ABB RobotStudio station: p3_robotstudio_2parte_ampliacion.rspag

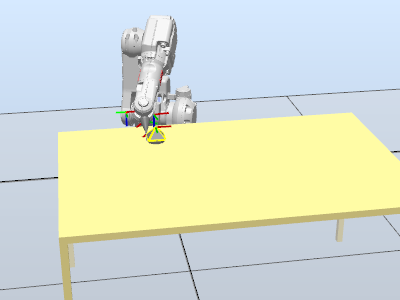
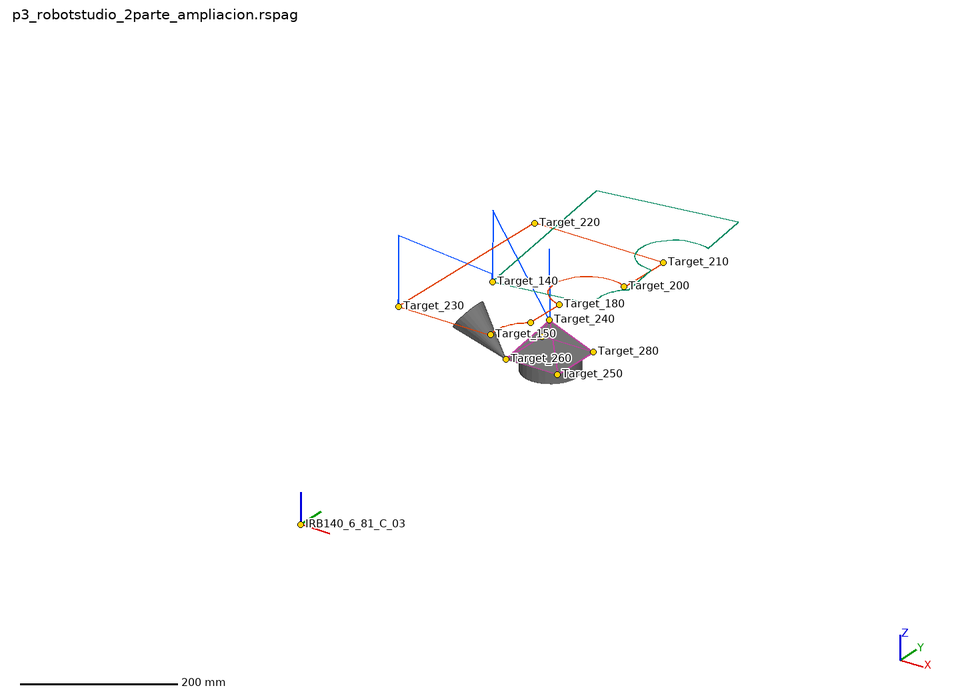
[picture v1: parts stored in the station drawn from their meshes, with robot base, taught points and paths (robot models come from the ABB library and are not in the file)]
--- station ---
Station p3_robotstudio_2parte (saved by RobotStudio 22.2.10013.1)
Controller Controlador1
  mechanical unit ROB_1: IRB140_6_81_C_03, 6 joints, base frame (0, 0, 0) mm
Layout (positions relative to the parent item):
  - printbed_hemisphere_hexagono [part, from Libraries\hemisphere.rslib] at (471.3, 85, 364.75) mm, rotated rx 90 ry 0 rz 0 deg
  - Mesa de trabajo [part, from Libraries\Mesa de trabajoDISA.rslib] at (1242.15, -525.68, -395) mm, rotated rx 0 ry 0 rz 90 deg
  - Pieza1 [part, from Libraries\Pieza_ampliacion.rslib] at (500, 0, 200) mm, rotated rx 0 ry 0 rz 90 deg
  - trazador [smart component, from Libraries\trazador.rslib] at (335.01, -108.97, 433.65) mm, rotated rx -146.48 ry 41.47 rz -135 deg
      connections:
        trazador.entrada_inyector -> TraceTCP.Enabled
        trazador.entrada_inyector -> ?.InputA
        ?.Output -> TraceTCP.Clear
    - TraceTCP [smart component, from Components\TraceTCP.rslib]
        properties: Robot=IRB140_6_81_C_03
  - IRB140_6_81_C_03 [mechanism, from Robots\IRB140_6_81_C_G_03.rslib] at (0, 0, 0) mm; joint values [-0.3661, -0.187, 0.842, 1.3893, 0.2881, -2.1751] (rad or m)
  - tool_laser [part] at (335.01, -108.97, 433.65) mm, rotated rx -146.48 ry 41.47 rz -135 deg, size 50 x 49.9 x 75 mm
  - tool_laser [mechanism] at (335.01, -108.97, 433.65) mm, rotated rx -146.48 ry 41.47 rz -135 deg
      TCP tool_laser at (0, 0, 75) mm
      links: Pieza_1
  - Curve_thing [part, from Training Objects\Curve_Thing.rslib] at (542.09, -125.55, 364.72) mm, rotated rx 0 ry 0.37 rz 89.92 deg
  - Pieza_4 [part] at (610.67, 44.58, 426.77) mm
  - Pieza_8 [part] at (-348.26, -126.32, -48.58) mm, size 80.8 x 80.4 x 70 mm
Attachment: trazador is attached to IRB140_6_81_C_03 / Link6
Attachment: tool_laser is attached to IRB140_6_81_C_03 / Link6
Attachment: tool_laser is attached to IRB140_6_81_C_03 / Link6
Attachment: Curve_thing is attached to Mesa de trabajo
Station logic (signal -> signal, property => property):
  Controlador1.activar_mecanizado -> trazador.entrada_inyector
Targets, tools, work objects and paths stored in the station and not in the controller backup, written as RAPID:
! task T_ROB1
MODULE Module1
  CONST robtarget Target_300:=[[-0.030300341,0.033376716,-0.180784391],[0.786632811,0.381173416,0.211660446,-0.437167591],[0,0,0,0],[9E+09,9E+09,9E+09,9E+09,9E+09,9E+09]];
ENDMODULE


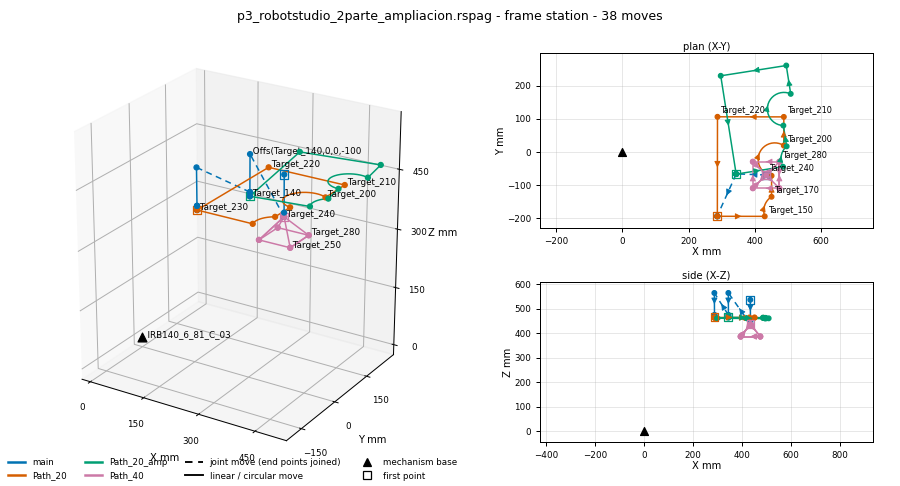
[picture p0: tool path of p3_robotstudio_2parte_ampliacion.rspag in frame station, 38 of 38 moves have a stored position in this frame; points joined in program order, loops and branches not executed]
--- Backups/Controlador1/RAPID/TASK1/PROGMOD/CalibData.mod ---
MODULE CalibData
    PERS tooldata tool_laser:=[TRUE,[[0,0,75],[1,0,0,0]],[1,[0,0,1],[1,0,0,0],0,0,0]];
    TASK PERS wobjdata Workobject:=[FALSE,TRUE,"",[[0,0,0],[1,0,0,0]],[[286.627001811,-193.490730871,464.561998296],[0.002682563,0.707605914,0.706600086,0.001729967]]];
    TASK PERS wobjdata wobj_mecanizado:=[FALSE,TRUE,"",[[0,0,0],[1,0,0,0]],[[286.627001811,-193.490730871,464.561998296],[0.002682563,0.707605914,0.706600086,0.001729967]]];
    TASK PERS wobjdata wobj_mecanizado_amp:=[FALSE,TRUE,"",[[343.366876171,-66.270210985,464.681994893],[0.002429835,0.649979761,0.759944792,-0.002078163]],[[0,0,0],[1,0,0,0]]];
    TASK PERS wobjdata wobj_mecanizado_2:=[FALSE,TRUE,"",[[146.920726873,124.553339247,-27.948128115],[1,0,0,0]],[[286.627001811,-193.490730871,464.561998296],[0.002682563,0.707605914,0.706600086,0.001729967]]];
ENDMODULE

--- Backups/Controlador1/RAPID/TASK1/PROGMOD/MainModule.mod ---
MODULE MainModule
    VAR bool ampliacion:=TRUE; ! ampliacion:=FALSE; to have the original condition
    VAR bool mecanizado2:=TRUE;
	PROC main()
        IF mecanizado2=TRUE THEN
            MoveJ Offs(Target_240,0,0,-100),v100,z100,tool_laser\WObj:=wobj_mecanizado_2;
            MoveL Offs(Target_240,0,0,-10),v30,fine,tool_laser\WObj:=wobj_mecanizado_2;
            MoveL Target_240,v5,fine,tool_laser\WObj:=wobj_mecanizado_2;
            Path_40;

        ELSE

            IF ampliacion = TRUE THEN
                MoveJ Offs(Target_140,0,0,-100),v100,z100,tool_laser\WObj:=wobj_mecanizado_amp;
                MoveL Offs(Target_140,0,0,-10),v30,fine,tool_laser\WObj:=wobj_mecanizado_amp;
                MoveL Target_140,v5,fine,tool_laser\WObj:=wobj_mecanizado_amp;
                Path_20_amp;
                MoveL Offs(Target_140,0,0,-10),v30,fine,tool_laser\WObj:=wobj_mecanizado_amp;

            ELSE
                MoveJ Offs(Target_140,0,0,-100),v100,z100,tool_laser\WObj:=wobj_mecanizado;
                MoveL Offs(Target_140,0,0,-10),v30,fine,tool_laser\WObj:=wobj_mecanizado;
                MoveL Target_140,v5,fine,tool_laser\WObj:=wobj_mecanizado;
                Path_20;
                MoveL Offs(Target_140,0,0,-10),v30,fine,tool_laser\WObj:=wobj_mecanizado;

            ENDIF
        ENDIF

    ENDPROC
ENDMODULE

--- Backups/Controlador1/RAPID/TASK1/PROGMOD/Module1.mod ---
MODULE Module1

    CONST robtarget Target_140:=[[-0.001044518,0.001237331,-0.119945019],[0.707118807,0.00041804,-0.0039884,0.707083383],[0,0,0,0],[9E+09,9E+09,9E+09,9E+09,9E+09,9E+09]];
    CONST robtarget Target_150:=[[0.00386513,142.872007259,0.770403421],[0.707118807,0.00041804,-0.0039884,0.707083383],[0,0,0,0],[9E+09,9E+09,9E+09,9E+09,9E+09,9E+09]];
    CONST robtarget Target_160:=[[33.145326632,142.71973051,0.936803286],[0.986143735,0.0026539,-0.003006478,0.165844662],[0,0,0,0],[9E+09,9E+09,9E+09,9E+09,9E+09,9E+09]];
    CONST robtarget Target_170:=[[59.100802816,163.32684758,1.196283016],[0.875444758,0.001507495,-0.003716121,0.483301555],[0,0,0,0],[9E+09,9E+09,9E+09,9E+09,9E+09,9E+09]];
    CONST robtarget Target_180:=[[122.520192337,163.322672707,1.516495109],[0.999991959,0.003115824,-0.002524627,-0.000025048],[0,0,0,0],[9E+09,9E+09,9E+09,9E+09,9E+09,9E+09]];
    CONST robtarget Target_190:=[[190.312689625,126.331594958,1.628299126],[0.981718547,0.002578379,-0.003071491,0.190296119],[0,0,0,0],[9E+09,9E+09,9E+09,9E+09,9E+09,9E+09]];
    CONST robtarget Target_200:=[[213.534871513,199.983297206,2.204533414],[0.476705541,-0.000734056,-0.003942493,0.879053892],[0,0,0,0],[9E+09,9E+09,9E+09,9E+09,9E+09,9E+09]];
    CONST robtarget Target_210:=[[300.002003583,199.97760511,2.641116318],[0.999991959,0.003115824,-0.002524627,-0.000025048],[0,0,0,0],[9E+09,9E+09,9E+09,9E+09,9E+09,9E+09]];
    CONST robtarget Target_220:=[[299.995130863,-0.018511296,1.394771596],[0.707083383,0.0039884,0.00041804,-0.707118807],[0,0,0,0],[9E+09,9E+09,9E+09,9E+09,9E+09,9E+09]];
    CONST robtarget Target_230:=[[-0.001044518,0.001237331,-0.119945019],[0.000025048,-0.002524627,-0.003115824,0.999991959],[0,0,0,0],[9E+09,9E+09,9E+09,9E+09,9E+09,9E+09]];
    CONST robtarget Target_240:=[[-0.030300341,0.033376716,-0.180784391],[0.247614936,0.417854629,0.116544073,0.866315088],[-1,0,-2,0],[9E+09,9E+09,9E+09,9E+09,9E+09,9E+09]];
    CONST robtarget Target_250:=[[-39.906344128,39.777551947,50.121834111],[0.247614936,0.417854629,0.116544073,0.866315088],[-1,0,-2,0],[9E+09,9E+09,9E+09,9E+09,9E+09,9E+09]];
    CONST robtarget Target_260:=[[-40.020477159,-40.221456481,49.622688614],[0.637610947,-0.304530712,0.308943455,-0.636606054],[0,0,0,0],[9E+09,9E+09,9E+09,9E+09,9E+09,9E+09]];
    CONST robtarget Target_270:=[[-0.030300341,0.033376716,-0.180784391],[0.865923454,0.122542991,0.416134867,0.248981041],[0,0,0,0],[9E+09,9E+09,9E+09,9E+09,9E+09,9E+09]];
    CONST robtarget Target_280:=[[40.09414935,39.664091458,50.013704819],[0.867229378,-0.116801792,-0.416517624,0.246543335],[0,0,0,0],[9E+09,9E+09,9E+09,9E+09,9E+09,9E+09]];
    CONST robtarget Target_290:=[[-39.906344128,39.777551947,50.121834111],[0.000932822,0.000299012,-0.435996822,0.899947672],[-1,-1,-2,0],[9E+09,9E+09,9E+09,9E+09,9E+09,9E+09]];
    CONST robtarget Target_310:=[[40.09414935,39.664091458,50.013704819],[0.787537393,0.381463377,-0.21113742,0.435535918],[0,0,0,0],[9E+09,9E+09,9E+09,9E+09,9E+09,9E+09]];
    CONST robtarget Target_320:=[[39.980016319,-40.33491697,49.514559322],[0.636112149,0.307649164,-0.304107845,-0.638930156],[0,0,0,0],[9E+09,9E+09,9E+09,9E+09,9E+09,9E+09]];
    CONST robtarget Target_330:=[[-0.030300341,0.033376716,-0.180784391],[0.437967882,-0.207871455,0.376843126,0.789279957],[0,0,0,0],[9E+09,9E+09,9E+09,9E+09,9E+09,9E+09]];
    CONST robtarget Target_340:=[[-40.020477159,-40.221456481,49.622688614],[0.437356992,-0.209472307,-0.37595563,-0.789618628],[-1,0,-2,0],[9E+09,9E+09,9E+09,9E+09,9E+09,9E+09]];
    CONST robtarget Target_350:=[[39.980016319,-40.33491697,49.514559322],[0.902650871,-0.43037245,0.000915201,-0.000349243],[1,-2,0,6],[9E+09,9E+09,9E+09,9E+09,9E+09,9E+09]];

    PROC Path_20()
        MoveL Target_140,v10,fine,tool_laser\WObj:=wobj_mecanizado;
        MoveL Target_150,v10,fine,tool_laser\WObj:=wobj_mecanizado;
        MoveC Target_160,Target_170,v10,fine,tool_laser\WObj:=wobj_mecanizado;
        MoveL Target_180,v10,fine,tool_laser\WObj:=wobj_mecanizado;
        MoveC Target_190,Target_200,v10,fine,tool_laser\WObj:=wobj_mecanizado;
        MoveL Target_210,v10,fine,tool_laser\WObj:=wobj_mecanizado;
        MoveL Target_220,v10,fine,tool_laser\WObj:=wobj_mecanizado;
        MoveL Target_230,v10,fine,tool_laser\WObj:=wobj_mecanizado;
    ENDPROC

    PROC Path_20_amp()
        MoveL Target_140,v10,fine,tool_laser\WObj:=wobj_mecanizado_amp;
        MoveL Target_150,v10,fine,tool_laser\WObj:=wobj_mecanizado_amp;
        MoveC Target_160,Target_170,v10,fine,tool_laser\WObj:=wobj_mecanizado_amp;
        MoveL Target_180,v10,fine,tool_laser\WObj:=wobj_mecanizado_amp;
        MoveC Target_190,Target_200,v10,fine,tool_laser\WObj:=wobj_mecanizado_amp;
        MoveL Target_210,v10,fine,tool_laser\WObj:=wobj_mecanizado_amp;
        MoveL Target_220,v10,fine,tool_laser\WObj:=wobj_mecanizado_amp;
        MoveL Target_230,v10,fine,tool_laser\WObj:=wobj_mecanizado_amp;
    ENDPROC
    PROC Path_40()
        MoveL Target_240,v10,fine,tool_laser\WObj:=wobj_mecanizado_2;
        MoveL Target_250,v10,fine,tool_laser\WObj:=wobj_mecanizado_2;
        MoveL Target_260,v10,fine,tool_laser\WObj:=wobj_mecanizado_2;
        MoveL Target_270,v10,fine,tool_laser\WObj:=wobj_mecanizado_2;
        MoveL Target_280,v10,fine,tool_laser\WObj:=wobj_mecanizado_2;
        MoveL Target_290,v10,fine,tool_laser\WObj:=wobj_mecanizado_2;
        MoveL Target_310,v10,fine,tool_laser\WObj:=wobj_mecanizado_2;
        MoveL Target_320,v10,fine,tool_laser\WObj:=wobj_mecanizado_2;
        MoveL Target_330,v10,fine,tool_laser\WObj:=wobj_mecanizado_2;
        MoveL Target_340,v10,fine,tool_laser\WObj:=wobj_mecanizado_2;
        MoveL Target_350,v10,fine,tool_laser\WObj:=wobj_mecanizado_2;
    ENDPROC
ENDMODULE

--- Backups/Controlador1/SYSPAR/EIO.cfg ---
EIO:CFG_1.0:6:1::
#
EIO_SIGNAL:

      -Name "activar_mecanizado" -SignalType "DO" -Access "All"
